Staubli VAL3: Form_PanelJoint.pgx

public program Form_PanelJoint(string x_sTitle, string x_sPanelTitle, jointRs& x_jJ[], num& x_nSelectIndex, string x_sBottom)
  local num l_nNum
begin

//×××××××××××××××××××××××××××××××××××××××××××××××××
//×××××××××××××××××××××××××××××××××××××××××××××××××
//if size(x_bList)!=size(x_sList)
//  return
//endIf
resize(sBuff,1,size(x_jJ))

for l_nNum=0 to size(sBuff)-1
//  if x_bList[l_nNum]
//    sBuff[l_nNum]=toString("",l_nNum+1)+"."+x_sList[l_nNum]
//  else
    sBuff[l_nNum]=toString("",l_nNum+1)+"."+"Joint"
//  endIf
endFor
//*********************************************************
call Form_PanelList(x_sTitle,x_sPanelTitle,sBuff,x_nSelectIndex,x_sBottom)

cls()

end
